(* Logix 5000 project; controller cal1615 1756-L62 rev 20.19; software revision 20.05; part 17 of 82 *)
(* tags used below, declared in another part *)
   FAULT : BOOL;   // Fault AFI
   p01_param_temp_limit : REAL;   // Machine Parameter Maximum Temperature for Fan Operation
   p01_sys_scp : SYS_SCP;   // System Scaling
   p01r02 : routine;   // System Misc Control
   p01r09_pb_global_reset : BOOL;   // System Modes PB: Global Fault Reset
   p11_ai_exh_amps : REAL;   // Zone 1 Analog Input Exhaust Fan Amps
   p11_ai_exh_hz : REAL;   // Zone 1 Analog Input Exhaust Fan HZ
   p11_ai_exh_hz_max : REAL;   // Zone 1 Analog Inputs Exhaust VFD max Hz
   p11_ai_exh_rpm : REAL;   // Zone 1 Analog Input Exhaust Fan RPM
   p11_ai_lfl : REAL;   // Zone 1 Analog Input Lower Flash Limit
   p11_ai_prs : REAL;   // Zone 1 Analog Input Pressure
   p11_ai_recirc_amps : REAL;   // Zone 1 Analog Input Recirc Fan Amps
   p11_ai_recirc_hz : REAL;   // Zone 1 Analog Input Supply Fan HZ
   p11_ai_recirc_hz_max : REAL;   // Zone 1 Analog Inputs Recric Fan Max Hz
   p11_ai_recirc_rpm : REAL;   // Zone 1 Analog Input Recirc Fan RPM
   p11_ai_tc01 : REAL;   // Zone 1 Analog Input Control Thermocouple 1
   p11_ai_tc02 : REAL;   // Zone 1 Analog Input Control Thermocouple 2
   p11_ao_cv : REAL;   // Zone 1 Analog Output Control Valve
   p11_ao_exhaust_selected_speed : REAL;   // Zone 1 Analog Output Exhaust Fan VFD Selected Speed
   p11_ao_recirc_selected_speed : REAL;   // Zone 1 Analog Output Recirc Fan VFD Selected Speed
   p11_di_burner_auto : BOOL;   // Zone 1 Digital Input Burner Auto
   p11_di_burner_safeties_ok : BOOL;   // Zone 1 Digital Input Burner Safeties Ok
   p11_di_door_open : BOOL;   // Zone 1 Digital Input Access Door Open
   p11_di_exh : acs800_di_normal;   // Zone 1 Digital Inputs Exhaust Fan
   p11_di_exh_fan_mtr_ts : BOOL;   // Zone 1 Digital Input Exhaust Fan Motor Thermostat OK
   p11_di_exh_flow_ok : BOOL;   // Zone 1 Digital Input Exhaust Flow OK
   p11_di_flame_failure : BOOL;   // Zone 1 Digital Input Flame Failure
   p11_di_flame_on : BOOL;   // Zone 1 Digital Input Burner is On
   p11_di_fresh_air_clean : BOOL;   // Zone 1 Digital Input Fresh Air Filter Dirty
   p11_di_high_limit_temp_ok : BOOL;   // Zone 1 Digital Input High Limit Temperature OK
   p11_di_recirc : acs800_di_normal;   // Zone 1 Digital Inputs Recirc Fan
   p11_di_recirc_fan_mtr_ts : BOOL;   // Zone 1 Digital Input Recirc Fan Motor Thermostat OK
   p11_di_recirc_flow_ok : BOOL;   // Zone 1 Digital Input Recirc Flow OK
   p11_di_sp0 : BOOL;   // Zone 1 Digital Input Combustion Blower Pressure OK
   p11_di_sp00 : BOOL;   // Zone 1 Digital Input Recirculation Air Filter Dirty
   p11_di_sp1 : BOOL;
   p11_di_sp2 : BOOL;
   p11_di_sp3 : BOOL;
   p11_di_tc01_bo : BOOL;   // Zone 1 Digital Input Control Thermocouple 1 Failure
   p11_di_tc02_bo : BOOL;   // Zone 1 Digital Input Control Thermocouple 2 Failure
   p11_di_zone_air_clean : BOOL;   // Zone 1 Digital Input Combustion Air Filter Dirty
   p11_dint_to_hmi : DINT[16];   // Zone 1 Temperature Control VFDs On
   p11_do_enable_burner : BOOL;   // Zone 1 Digital Output Enable Burner
   p11_do_exh : acs800_do_normal;   // Zone 1 Digital Output Exhaust Fan
   p11_do_recirc : acs800_do_normal;   // Zone 1 Digital Outputs Supply Fan
   p11_do_rst_flame : BOOL;   // Zone 1 Digital Output Reset Flame Safety
   p11_exhaust_input_max : REAL;
   p11_exhaust_input_min : REAL;   // Zone 1 Exhaust Input Minimum
   p11_exhaust_output_max : REAL;
   p11_exhaust_output_min : REAL;
   p11_hc_input_max : REAL;
   p11_hc_input_min : REAL;
   p11_hc_output_max : REAL;
   p11_hc_output_min : REAL;
   p11_lfl_input_max : REAL;
   p11_lfl_input_min : REAL;
   p11_lfl_output_max : REAL;
   p11_lfl_output_min : REAL;
   p11_param_shutdown_temp : REAL;   // Zone 1 Parameter Zone Shutdown Temperature
   p11_param_tc01z : REAL;   // Zone 1 Parameter Process Temperature Zero Offset
   p11_param_tc02z : REAL;   // Zone 1 Parameter SupplyTemperature Zero Offset
   p11_param_zone_pressure : REAL;   // Zone 1 Parameter High Pressure LImit
   p11_prs_input_max : REAL;
   p11_prs_input_min : REAL;
   p11_prs_output_max : REAL;
   p11_prs_output_min : REAL;
   p11_recirc_input_max : REAL;
   p11_recirc_input_min : REAL;
   p11_recirc_output_max : REAL;
   p11_recirc_output_min : REAL;
   p11r01 : routine;   // Zone 1 Main
   p11r02 : routine;   // Zone 1 Misc Control
   p11r02_fault_exists : BOOL;
   p11r02_not_safe_temp : BOOL;   // Zone 1 Misc Control Zone above Safe Temp
   p11r02_safe_temp : BOOL;   // Zone 1 Misc Control Zone Temperature at Safe Temp
   p11r02_shutdown_temp : BOOL;   // Zone 1 Misc Control Safe Shutdown Temperature
   p11r02_timer_fault : TIMER[4];   // Zone 1 Misc Control Fault Delay
   p11r02_timer_safe_temp : TIMER[2];   // Zone 1 Misc Control Chamber SafeTemperature Dwell
   p11r02_timer_warning : TIMER[4];   // Zone 1 Misc Control Warning Delay
   p11r02_unack_fault : BOOL;   // Zone 1 Misc Control Unacknowledged Fault Exists
   p11r02_unack_warning : BOOL;   // Zone 1 Misc Control Unacknowledged Warning Exists
   p11r02_warning_exists : BOOL;
   p11r03 : routine;   // Zone 1 Input
   p11r03_hz : SYS_SCP;   // Zone 1 Analog Inputs SCP Hz
   p11r03_timer_fault : TIMER[4];   // Zone 1 Input Fault Delay
   p11r03_timer_warning : TIMER[4];   // Zone 1 Input Warning Delay
   p11r04 : routine;   // Zone 1 Output
   p11r04_timer_fault : TIMER[4];   // Zone 1 Output Fault Delay
   p11r04_timer_warning : TIMER[4];   // Zone 1 Output Warning Delay
   p11r05 : routine;   // Zone 1 Dint to HMI
   p11r06 : routine;   // Zone 1 Real to HMI
   p11r07 : routine;   // Zone 1 Alarms
   p11r08 : routine;   // Zone 1 Warnings
   p11r09 : routine;   // Zone 1 Modes
   p11r10 : routine;   // Zone 1
   p11r20 : routine;   // Zone 1 Temp Sequence
   p11r30 : routine;   // Zone 1 Temperature Control
   p11r30_pb_zone_off : BOOL;   // Zone 1 Temperature Control PB: Stop Zone Heat Control
   p11r31 : routine;   // Zone 1 Exhaust VFD
   p11r32 : routine;   // Zone 1 Recirc VFD
(* P11_Zone_1, continued *)

ROUTINE R02_Misc_Control   (* ladder *)
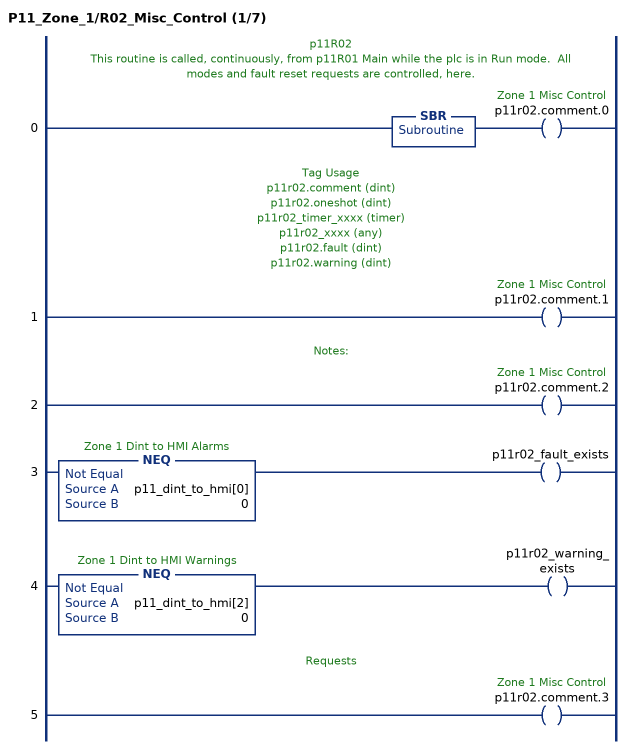
   // p11R02
   // This routine is called, continuously, from p11R01 Main while the plc is in Run mode.  All modes and fault reset requests are controlled, here.
   0: SBR()OTE(p11r02.comment.0);
   // Tag Usage
   // p11r02.comment (dint)
   // p11r02.oneshot (dint)
   // p11r02_timer_xxxx (timer)
   // p11r02_xxxx (any)
   // p11r02.fault (dint)
   // p11r02.warning (dint)
   1: OTE(p11r02.comment.1);
   // Notes:
   2: OTE(p11r02.comment.2);
   3: NEQ(p11_dint_to_hmi[0],0)OTE(p11r02_fault_exists);
   4: NEQ(p11_dint_to_hmi[2],0)OTE(p11r02_warning_exists);
   // Requests
   5: OTE(p11r02.comment.3);
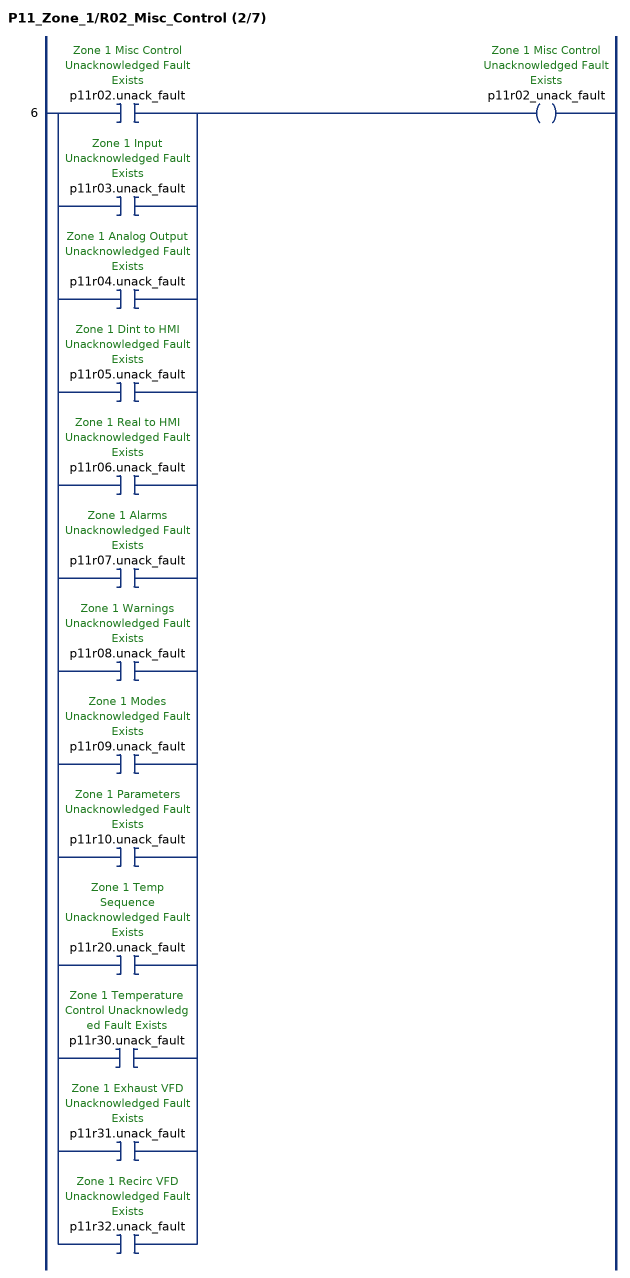
   6: [XIC(p11r02.unack_fault) ,XIC(p11r03.unack_fault) ,XIC(p11r04.unack_fault) ,XIC(p11r05.unack_fault) ,XIC(p11r06.unack_fault) ,XIC(p11r07.unack_fault) ,XIC(p11r08.unack_fault) ,XIC(p11r09.unack_fault) ,XIC(p11r10.unack_fault) ,XIC(p11r20.unack_fault) ,XIC(p11r30.unack_fault) ,XIC(p11r31.unack_fault) ,XIC(p11r32.unack_fault) ]OTE(p11r02_unack_fault);
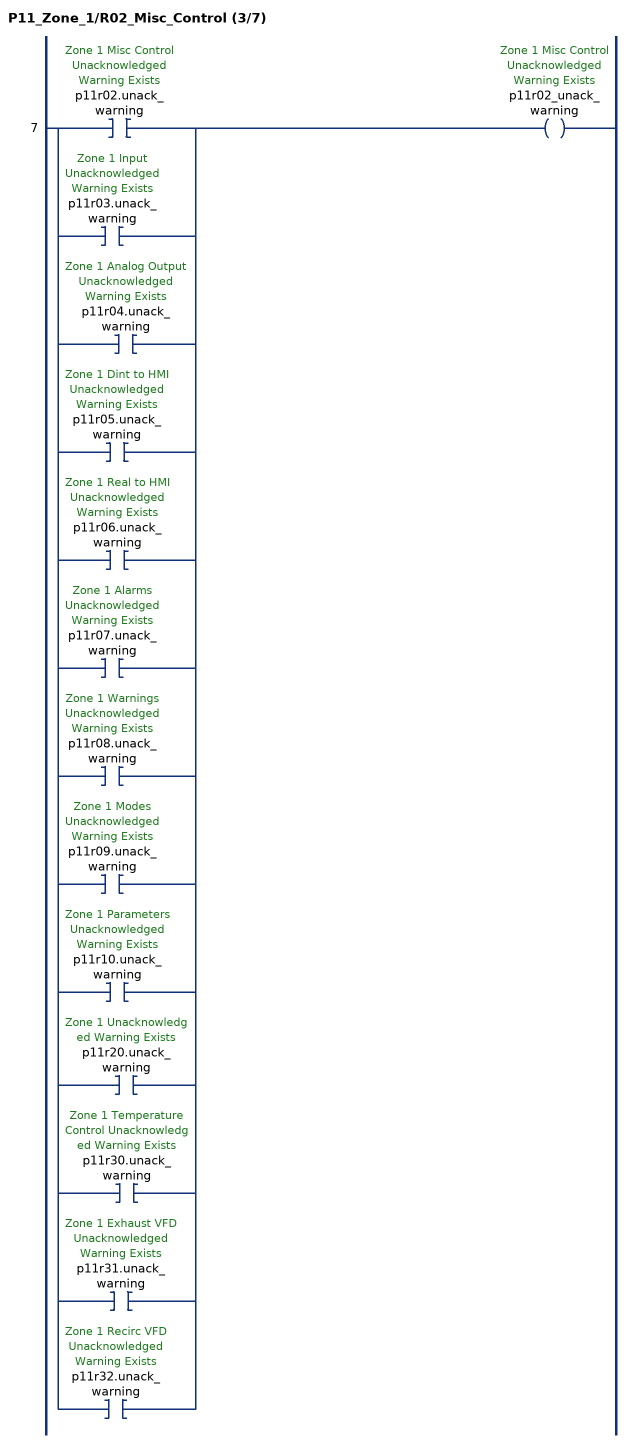
   7: [XIC(p11r02.unack_warning) ,XIC(p11r03.unack_warning) ,XIC(p11r04.unack_warning) ,XIC(p11r05.unack_warning) ,XIC(p11r06.unack_warning) ,XIC(p11r07.unack_warning) ,XIC(p11r08.unack_warning) ,XIC(p11r09.unack_warning) ,XIC(p11r10.unack_warning) ,XIC(p11r20.unack_warning) ,XIC(p11r30.unack_warning) ,XIC(p11r31.unack_warning) ,XIC(p11r32.unack_warning) ]OTE(p11r02_unack_warning);
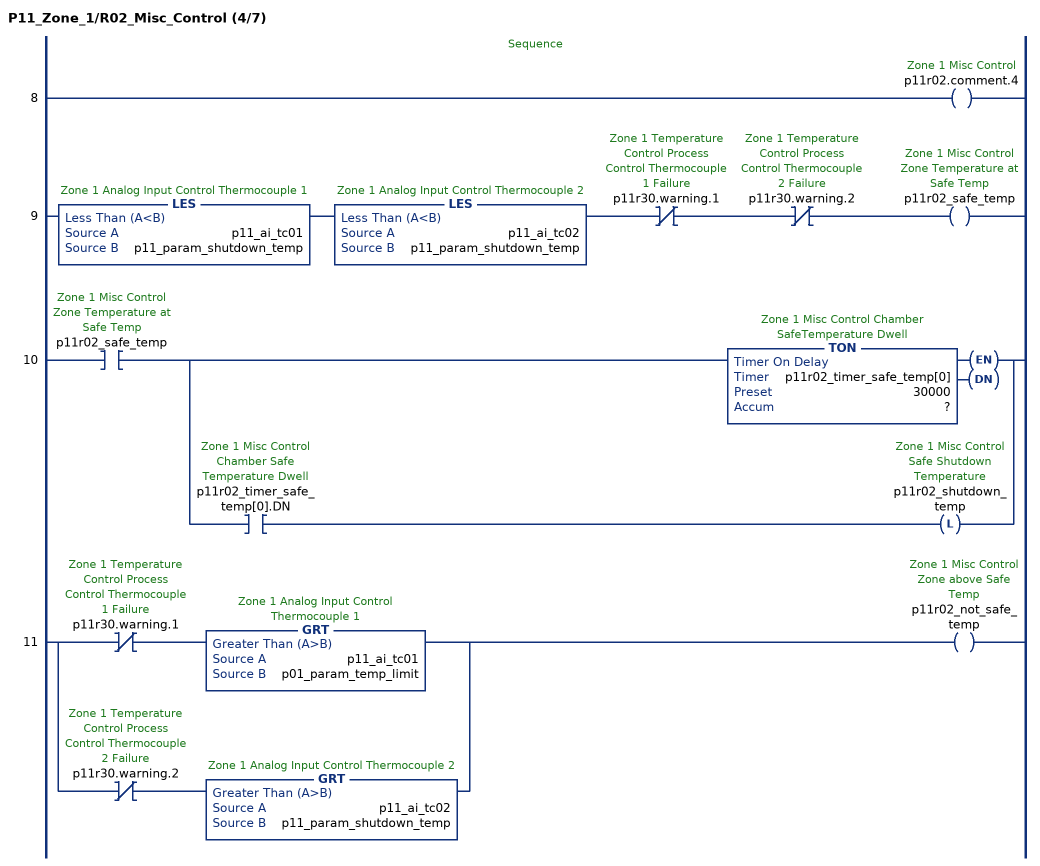
   // Sequence
   8: OTE(p11r02.comment.4);
   9: LES(p11_ai_tc01,p11_param_shutdown_temp)LES(p11_ai_tc02,p11_param_shutdown_temp)XIO(p11r30.warning.1)XIO(p11r30.warning.2)OTE(p11r02_safe_temp);
   10: XIC(p11r02_safe_temp)[TON(p11r02_timer_safe_temp[0],?,?) ,XIC(p11r02_timer_safe_temp[0].DN) OTL(p11r02_shutdown_temp) ];
   11: [XIO(p11r30.warning.1) GRT(p11_ai_tc01,p01_param_temp_limit) ,XIO(p11r30.warning.2) GRT(p11_ai_tc02,p11_param_shutdown_temp) ]OTE(p11r02_not_safe_temp);
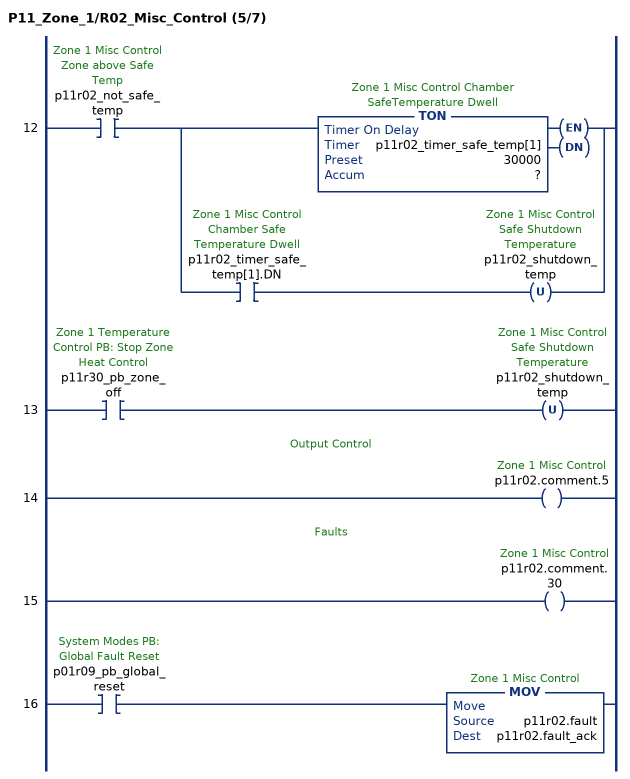
   12: XIC(p11r02_not_safe_temp)[TON(p11r02_timer_safe_temp[1],?,?) ,XIC(p11r02_timer_safe_temp[1].DN) OTU(p11r02_shutdown_temp) ];
   13: XIC(p11r30_pb_zone_off)OTU(p11r02_shutdown_temp);
   // Output Control
   14: OTE(p11r02.comment.5);
   // Faults
   15: OTE(p11r02.comment.30);
   16: XIC(p01r09_pb_global_reset)MOV(p11r02.fault,p11r02.fault_ack);
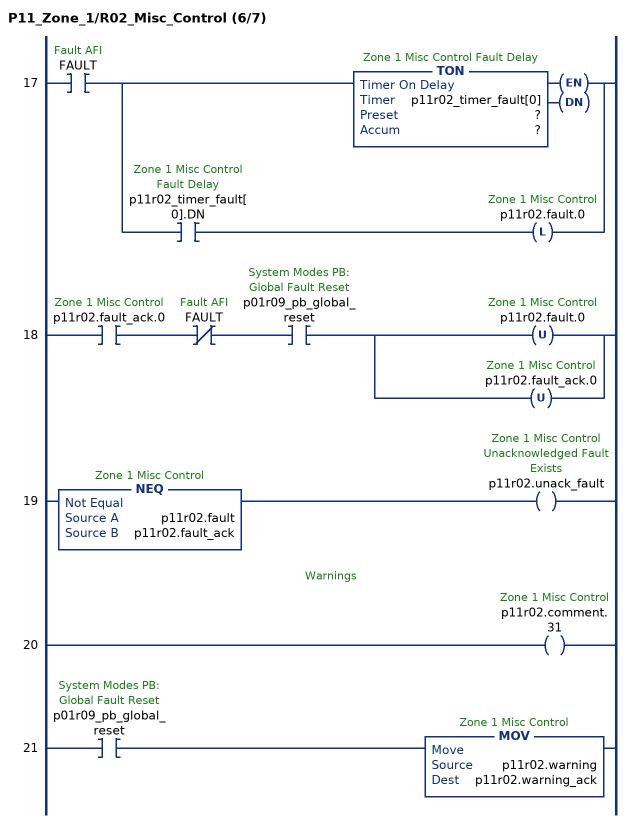
   17: XIC(FAULT)[TON(p11r02_timer_fault[0],?,?) ,XIC(p11r02_timer_fault[0].DN) OTL(p11r02.fault.0) ];
   18: XIC(p11r02.fault_ack.0)XIO(FAULT)XIC(p01r09_pb_global_reset)[OTU(p11r02.fault.0) ,OTU(p11r02.fault_ack.0) ];
   19: NEQ(p11r02.fault,p11r02.fault_ack)OTE(p11r02.unack_fault);
   // Warnings
   20: OTE(p11r02.comment.31);
   21: XIC(p01r09_pb_global_reset)MOV(p11r02.warning,p11r02.warning_ack);
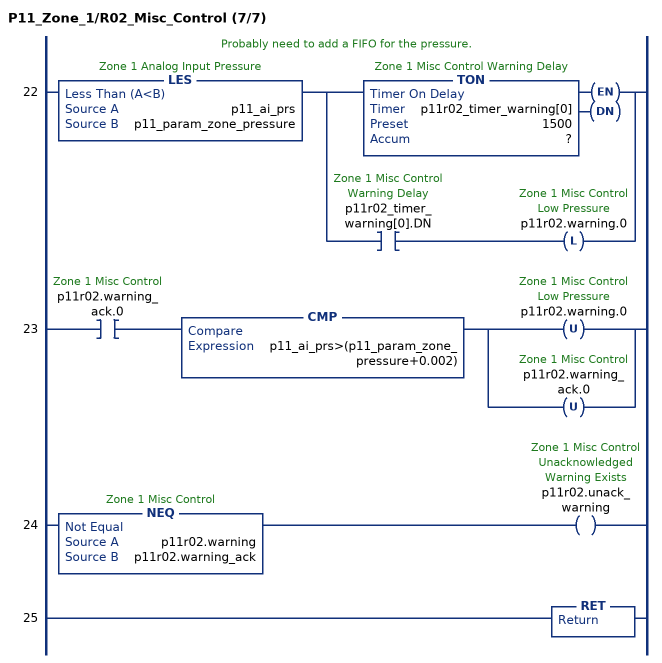
   // Probably need to add a FIFO for the pressure.
   22: LES(p11_ai_prs,p11_param_zone_pressure)[TON(p11r02_timer_warning[0],?,?) ,XIC(p11r02_timer_warning[0].DN) OTL(p11r02.warning.0) ];
   23: XIC(p11r02.warning_ack.0)CMP(p11_ai_prs>(p11_param_zone_pressure+0.002))[OTU(p11r02.warning.0) ,OTU(p11r02.warning_ack.0) ];
   24: NEQ(p11r02.warning,p11r02.warning_ack)OTE(p11r02.unack_warning);
   25: RET();
END_ROUTINE

ROUTINE R03_Input   (* ladder *)
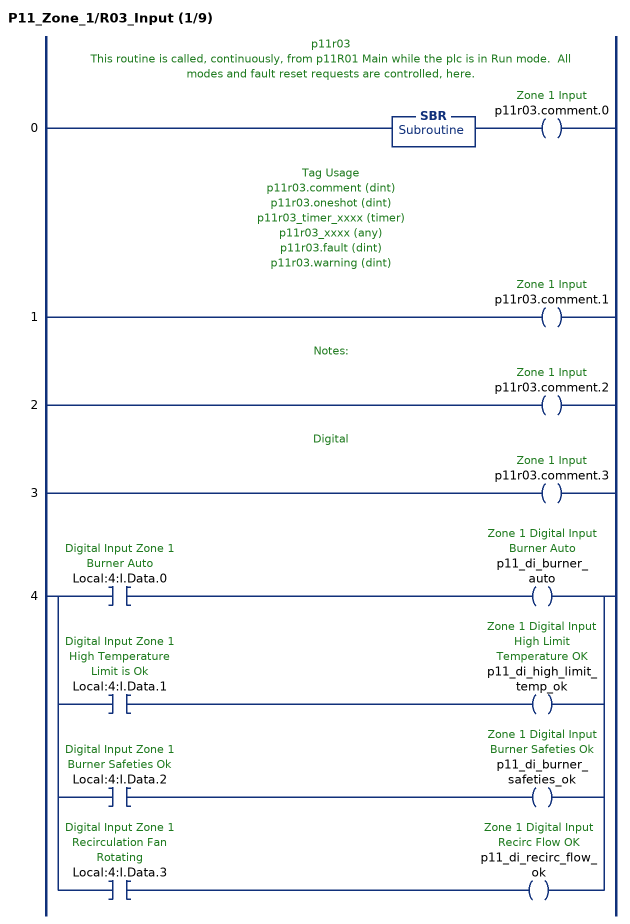
   // p11r03
   // This routine is called, continuously, from p11R01 Main while the plc is in Run mode.  All modes and fault reset requests are controlled, here.
   0: SBR()OTE(p11r03.comment.0);
   // Tag Usage
   // p11r03.comment (dint)
   // p11r03.oneshot (dint)
   // p11r03_timer_xxxx (timer)
   // p11r03_xxxx (any)
   // p11r03.fault (dint)
   // p11r03.warning (dint)
   1: OTE(p11r03.comment.1);
   // Notes:
   2: OTE(p11r03.comment.2);
   // Digital
   3: OTE(p11r03.comment.3);
   4: [XIC(Local:4:I.Data.0) OTE(p11_di_burner_auto) ,XIC(Local:4:I.Data.1) OTE(p11_di_high_limit_temp_ok) ,XIC(Local:4:I.Data.2) OTE(p11_di_burner_safeties_ok) ,XIC(Local:4:I.Data.3) OTE(p11_di_recirc_flow_ok) ];
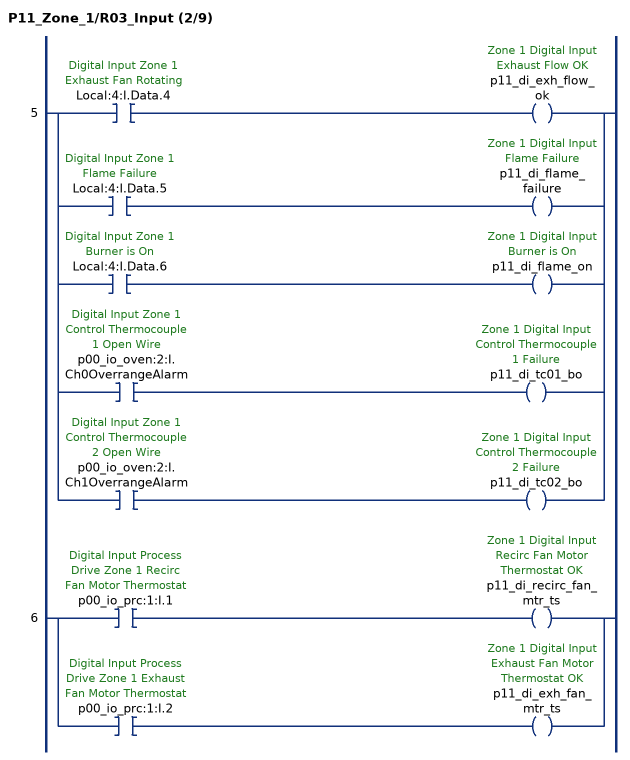
   5: [XIC(Local:4:I.Data.4) OTE(p11_di_exh_flow_ok) ,XIC(Local:4:I.Data.5) OTE(p11_di_flame_failure) ,XIC(Local:4:I.Data.6) OTE(p11_di_flame_on) ,XIC(p00_io_oven:2:I.Ch0OverrangeAlarm) OTE(p11_di_tc01_bo) ,XIC(p00_io_oven:2:I.Ch1OverrangeAlarm) OTE(p11_di_tc02_bo) ];
   6: [XIC(p00_io_prc:1:I.1) OTE(p11_di_recirc_fan_mtr_ts) ,XIC(p00_io_prc:1:I.2) OTE(p11_di_exh_fan_mtr_ts) ];
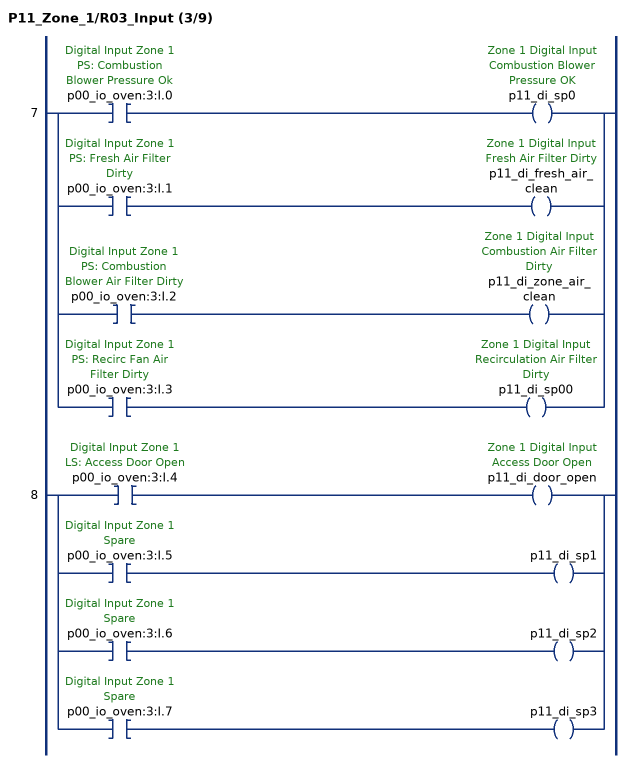
   7: [XIC(p00_io_oven:3:I.0) OTE(p11_di_sp0) ,XIC(p00_io_oven:3:I.1) OTE(p11_di_fresh_air_clean) ,XIC(p00_io_oven:3:I.2) OTE(p11_di_zone_air_clean) ,XIC(p00_io_oven:3:I.3) OTE(p11_di_sp00) ];
   8: [XIC(p00_io_oven:3:I.4) OTE(p11_di_door_open) ,XIC(p00_io_oven:3:I.5) OTE(p11_di_sp1) ,XIC(p00_io_oven:3:I.6) OTE(p11_di_sp2) ,XIC(p00_io_oven:3:I.7) OTE(p11_di_sp3) ];
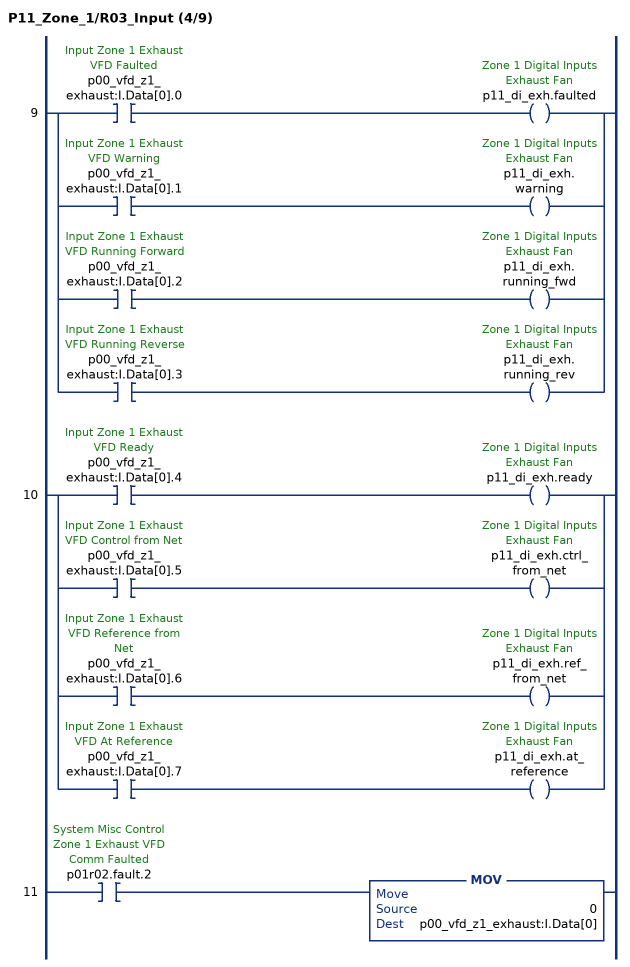
   9: [XIC(p00_vfd_z1_exhaust:I.Data[0].0) OTE(p11_di_exh.faulted) ,XIC(p00_vfd_z1_exhaust:I.Data[0].1) OTE(p11_di_exh.warning) ,XIC(p00_vfd_z1_exhaust:I.Data[0].2) OTE(p11_di_exh.running_fwd) ,XIC(p00_vfd_z1_exhaust:I.Data[0].3) OTE(p11_di_exh.running_rev) ];
   10: [XIC(p00_vfd_z1_exhaust:I.Data[0].4) OTE(p11_di_exh.ready) ,XIC(p00_vfd_z1_exhaust:I.Data[0].5) OTE(p11_di_exh.ctrl_from_net) ,XIC(p00_vfd_z1_exhaust:I.Data[0].6) OTE(p11_di_exh.ref_from_net) ,XIC(p00_vfd_z1_exhaust:I.Data[0].7) OTE(p11_di_exh.at_reference) ];
   11: XIC(p01r02.fault.2)MOV(0,p00_vfd_z1_exhaust:I.Data[0]);
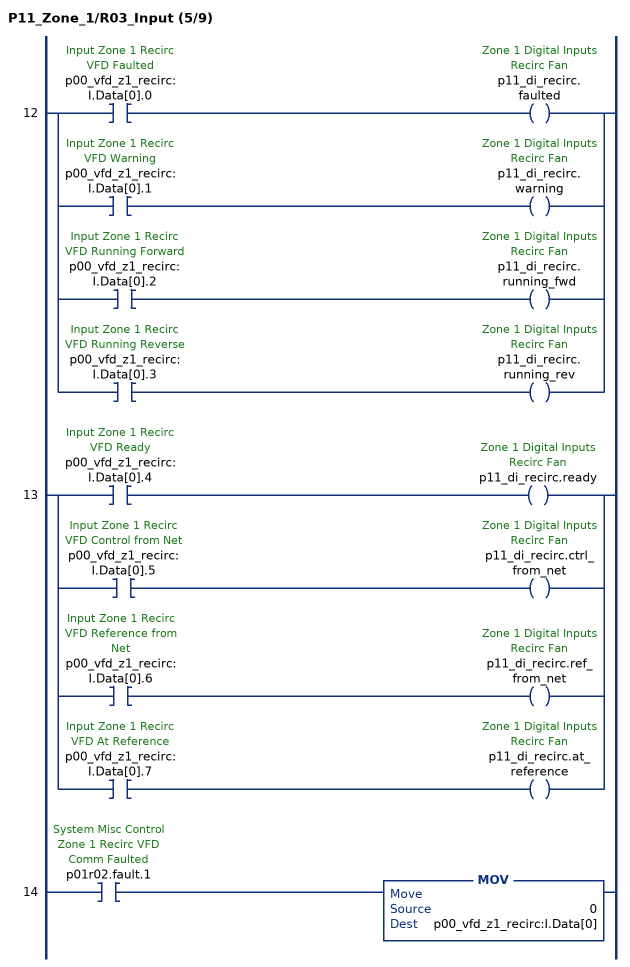
   12: [XIC(p00_vfd_z1_recirc:I.Data[0].0) OTE(p11_di_recirc.faulted) ,XIC(p00_vfd_z1_recirc:I.Data[0].1) OTE(p11_di_recirc.warning) ,XIC(p00_vfd_z1_recirc:I.Data[0].2) OTE(p11_di_recirc.running_fwd) ,XIC(p00_vfd_z1_recirc:I.Data[0].3) OTE(p11_di_recirc.running_rev) ];
   13: [XIC(p00_vfd_z1_recirc:I.Data[0].4) OTE(p11_di_recirc.ready) ,XIC(p00_vfd_z1_recirc:I.Data[0].5) OTE(p11_di_recirc.ctrl_from_net) ,XIC(p00_vfd_z1_recirc:I.Data[0].6) OTE(p11_di_recirc.ref_from_net) ,XIC(p00_vfd_z1_recirc:I.Data[0].7) OTE(p11_di_recirc.at_reference) ];
   14: XIC(p01r02.fault.1)MOV(0,p00_vfd_z1_recirc:I.Data[0]);
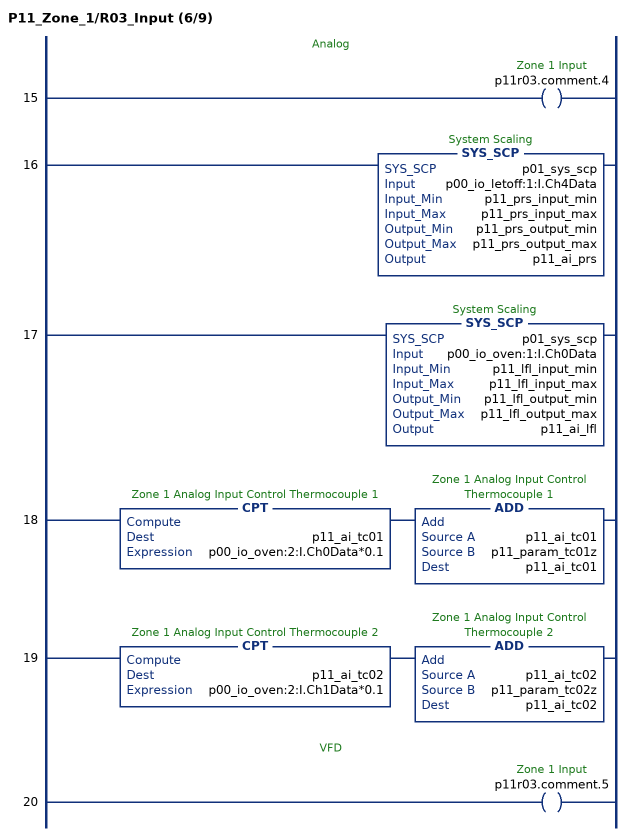
   // Analog
   15: OTE(p11r03.comment.4);
   16: SYS_SCP(p01_sys_scp,p00_io_letoff:1:I.Ch4Data,p11_prs_input_min,p11_prs_input_max,p11_prs_output_min,p11_prs_output_max,p11_ai_prs);
   17: SYS_SCP(p01_sys_scp,p00_io_oven:1:I.Ch0Data,p11_lfl_input_min,p11_lfl_input_max,p11_lfl_output_min,p11_lfl_output_max,p11_ai_lfl);
   18: CPT(p11_ai_tc01,p00_io_oven:2:I.Ch0Data*0.1)ADD(p11_ai_tc01,p11_param_tc01z,p11_ai_tc01);
   19: CPT(p11_ai_tc02,p00_io_oven:2:I.Ch1Data*0.1)ADD(p11_ai_tc02,p11_param_tc02z,p11_ai_tc02);
   // VFD
   20: OTE(p11r03.comment.5);
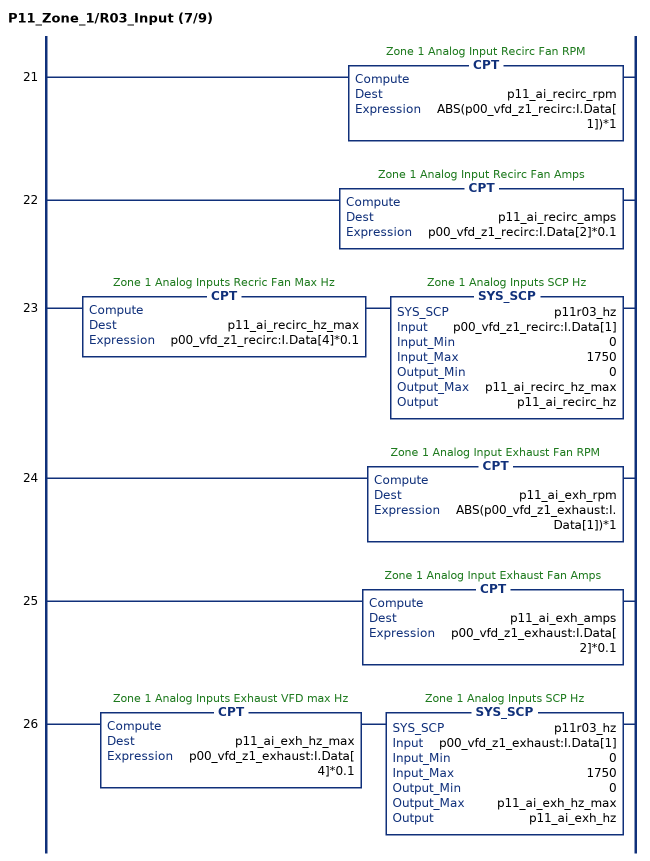
   21: CPT(p11_ai_recirc_rpm,ABS(p00_vfd_z1_recirc:I.Data[1])*1);
   22: CPT(p11_ai_recirc_amps,p00_vfd_z1_recirc:I.Data[2]*0.1);
   23: CPT(p11_ai_recirc_hz_max,p00_vfd_z1_recirc:I.Data[4]*0.1)SYS_SCP(p11r03_hz,p00_vfd_z1_recirc:I.Data[1],0,1750,0,p11_ai_recirc_hz_max,p11_ai_recirc_hz);
   24: CPT(p11_ai_exh_rpm,ABS(p00_vfd_z1_exhaust:I.Data[1])*1);
   25: CPT(p11_ai_exh_amps,p00_vfd_z1_exhaust:I.Data[2]*0.1);
   26: CPT(p11_ai_exh_hz_max,p00_vfd_z1_exhaust:I.Data[4]*0.1)SYS_SCP(p11r03_hz,p00_vfd_z1_exhaust:I.Data[1],0,1750,0,p11_ai_exh_hz_max,p11_ai_exh_hz);
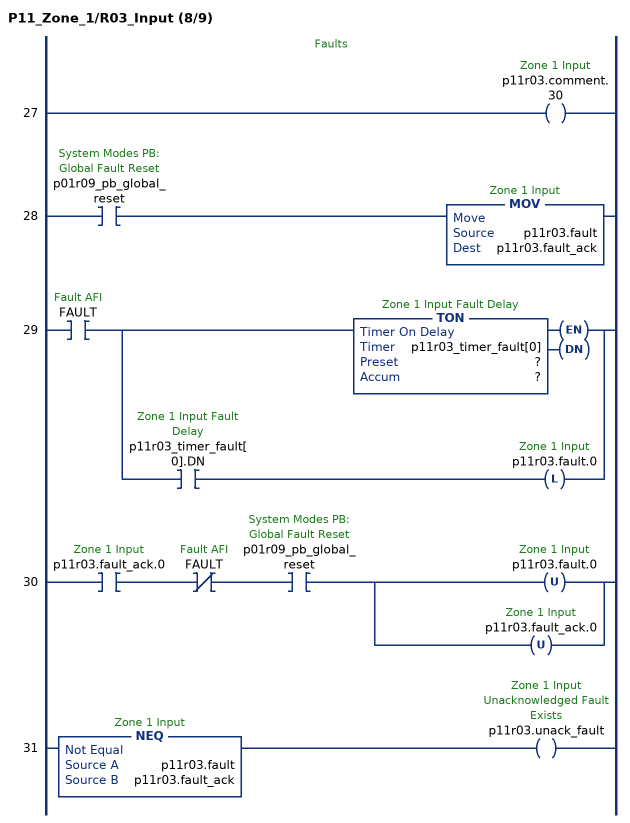
   // Faults
   27: OTE(p11r03.comment.30);
   28: XIC(p01r09_pb_global_reset)MOV(p11r03.fault,p11r03.fault_ack);
   29: XIC(FAULT)[TON(p11r03_timer_fault[0],?,?) ,XIC(p11r03_timer_fault[0].DN) OTL(p11r03.fault.0) ];
   30: XIC(p11r03.fault_ack.0)XIO(FAULT)XIC(p01r09_pb_global_reset)[OTU(p11r03.fault.0) ,OTU(p11r03.fault_ack.0) ];
   31: NEQ(p11r03.fault,p11r03.fault_ack)OTE(p11r03.unack_fault);
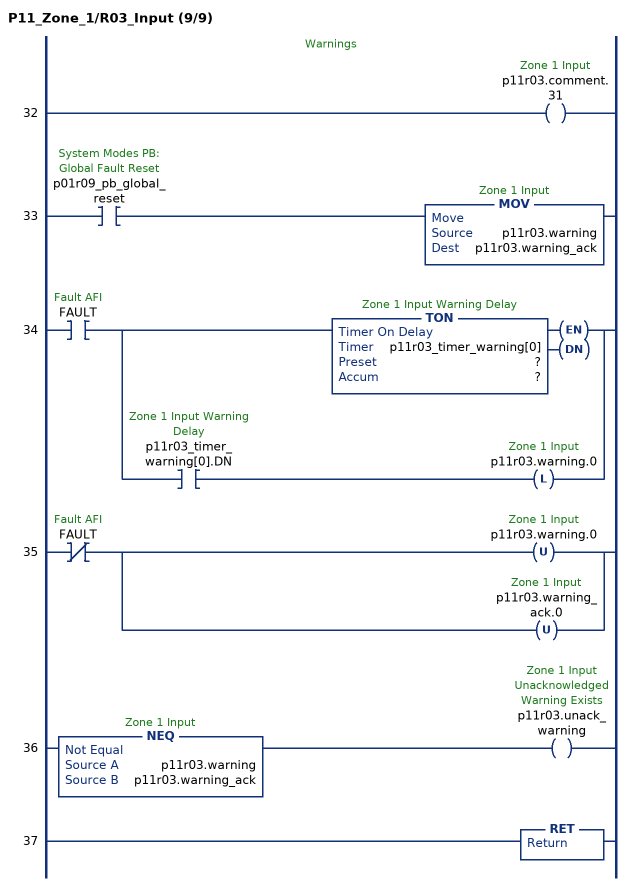
   // Warnings
   32: OTE(p11r03.comment.31);
   33: XIC(p01r09_pb_global_reset)MOV(p11r03.warning,p11r03.warning_ack);
   34: XIC(FAULT)[TON(p11r03_timer_warning[0],?,?) ,XIC(p11r03_timer_warning[0].DN) OTL(p11r03.warning.0) ];
   35: XIO(FAULT)[OTU(p11r03.warning.0) ,OTU(p11r03.warning_ack.0) ];
   36: NEQ(p11r03.warning,p11r03.warning_ack)OTE(p11r03.unack_warning);
   37: RET();
END_ROUTINE

ROUTINE R04_Output   (* ladder *)
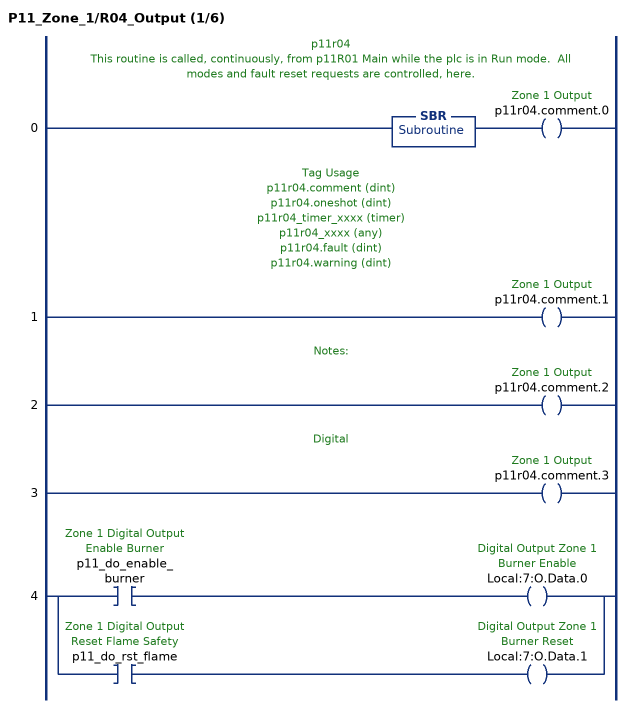
   // p11r04
   // This routine is called, continuously, from p11R01 Main while the plc is in Run mode.  All modes and fault reset requests are controlled, here.
   0: SBR()OTE(p11r04.comment.0);
   // Tag Usage
   // p11r04.comment (dint)
   // p11r04.oneshot (dint)
   // p11r04_timer_xxxx (timer)
   // p11r04_xxxx (any)
   // p11r04.fault (dint)
   // p11r04.warning (dint)
   1: OTE(p11r04.comment.1);
   // Notes:
   2: OTE(p11r04.comment.2);
   // Digital
   3: OTE(p11r04.comment.3);
   4: [XIC(p11_do_enable_burner) OTE(Local:7:O.Data.0) ,XIC(p11_do_rst_flame) OTE(Local:7:O.Data.1) ];
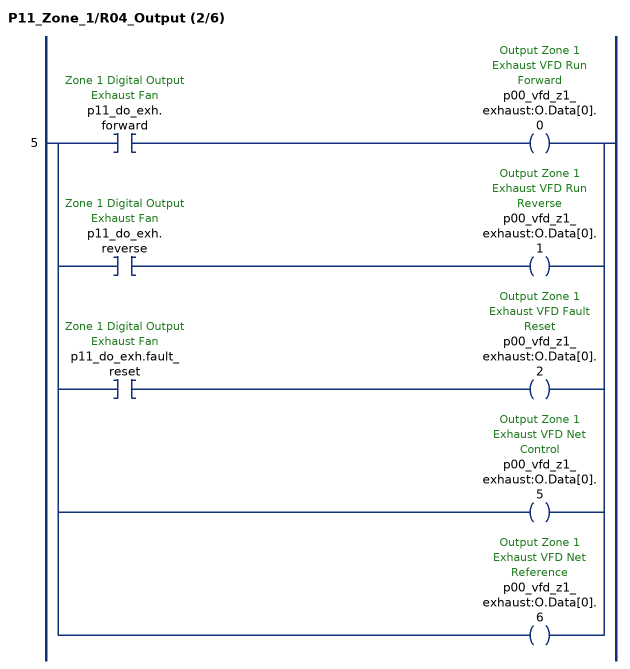
   5: [XIC(p11_do_exh.forward) OTE(p00_vfd_z1_exhaust:O.Data[0].0) ,XIC(p11_do_exh.reverse) OTE(p00_vfd_z1_exhaust:O.Data[0].1) ,XIC(p11_do_exh.fault_reset) OTE(p00_vfd_z1_exhaust:O.Data[0].2) ,OTE(p00_vfd_z1_exhaust:O.Data[0].5) ,OTE(p00_vfd_z1_exhaust:O.Data[0].6) ];
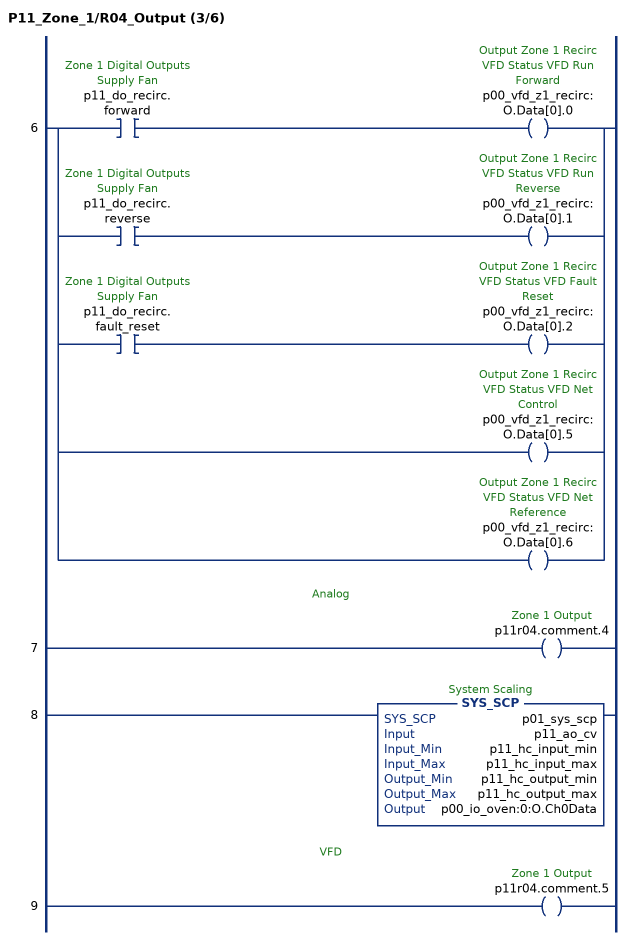
   6: [XIC(p11_do_recirc.forward) OTE(p00_vfd_z1_recirc:O.Data[0].0) ,XIC(p11_do_recirc.reverse) OTE(p00_vfd_z1_recirc:O.Data[0].1) ,XIC(p11_do_recirc.fault_reset) OTE(p00_vfd_z1_recirc:O.Data[0].2) ,OTE(p00_vfd_z1_recirc:O.Data[0].5) ,OTE(p00_vfd_z1_recirc:O.Data[0].6) ];
   // Analog
   7: OTE(p11r04.comment.4);
   8: SYS_SCP(p01_sys_scp,p11_ao_cv,p11_hc_input_min,p11_hc_input_max,p11_hc_output_min,p11_hc_output_max,p00_io_oven:0:O.Ch0Data);
   // VFD
   9: OTE(p11r04.comment.5);
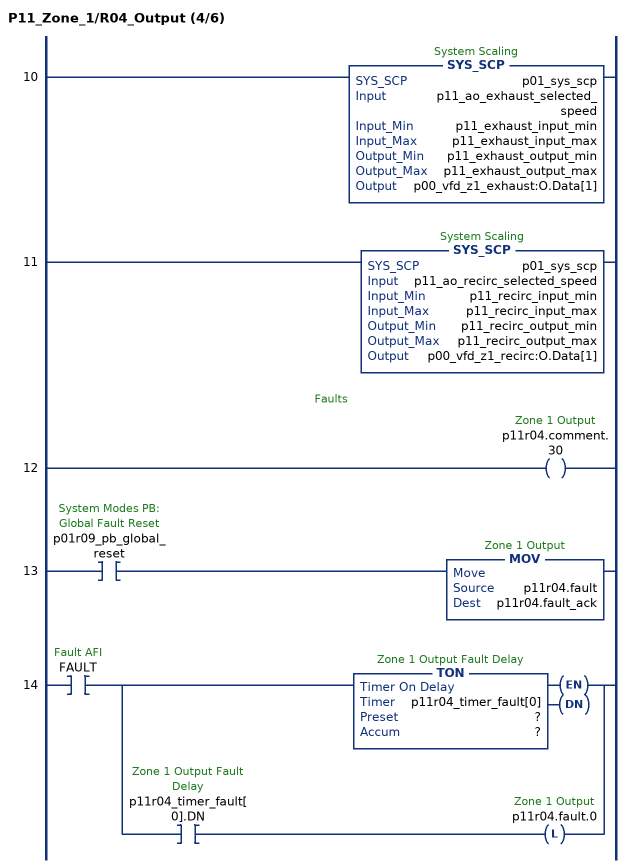
   10: SYS_SCP(p01_sys_scp,p11_ao_exhaust_selected_speed,p11_exhaust_input_min,p11_exhaust_input_max,p11_exhaust_output_min,p11_exhaust_output_max,p00_vfd_z1_exhaust:O.Data[1]);
   11: SYS_SCP(p01_sys_scp,p11_ao_recirc_selected_speed,p11_recirc_input_min,p11_recirc_input_max,p11_recirc_output_min,p11_recirc_output_max,p00_vfd_z1_recirc:O.Data[1]);
   // Faults
   12: OTE(p11r04.comment.30);
   13: XIC(p01r09_pb_global_reset)MOV(p11r04.fault,p11r04.fault_ack);
   14: XIC(FAULT)[TON(p11r04_timer_fault[0],?,?) ,XIC(p11r04_timer_fault[0].DN) OTL(p11r04.fault.0) ];
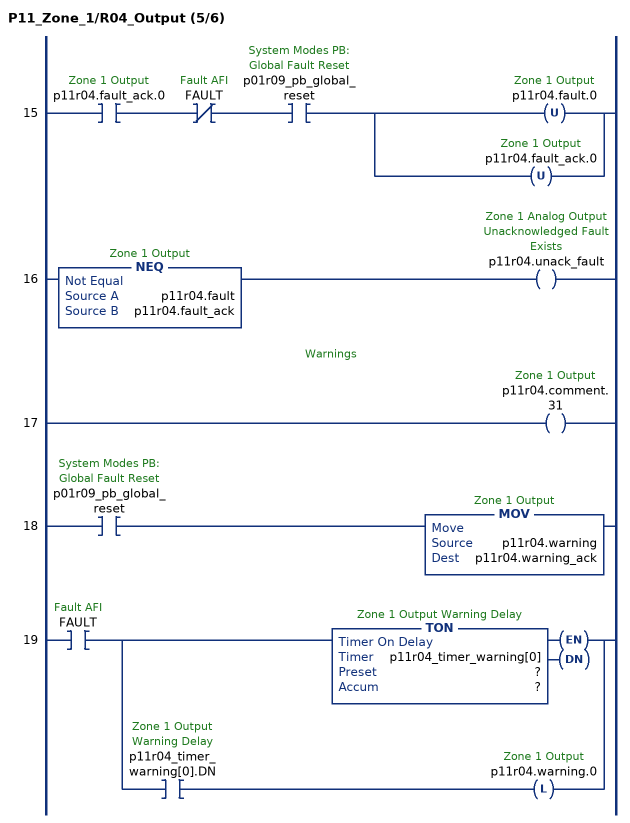
   15: XIC(p11r04.fault_ack.0)XIO(FAULT)XIC(p01r09_pb_global_reset)[OTU(p11r04.fault.0) ,OTU(p11r04.fault_ack.0) ];
   16: NEQ(p11r04.fault,p11r04.fault_ack)OTE(p11r04.unack_fault);
   // Warnings
   17: OTE(p11r04.comment.31);
   18: XIC(p01r09_pb_global_reset)MOV(p11r04.warning,p11r04.warning_ack);
   19: XIC(FAULT)[TON(p11r04_timer_warning[0],?,?) ,XIC(p11r04_timer_warning[0].DN) OTL(p11r04.warning.0) ];
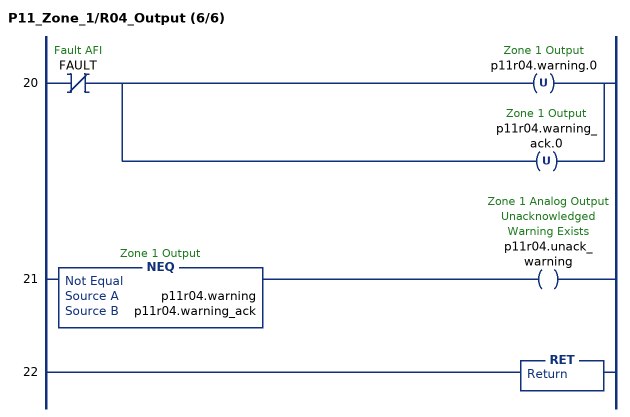
   20: XIO(FAULT)[OTU(p11r04.warning.0) ,OTU(p11r04.warning_ack.0) ];
   21: NEQ(p11r04.warning,p11r04.warning_ack)OTE(p11r04.unack_warning);
   22: RET();
END_ROUTINE
